FUNCTION_BLOCK PUBLIC FB_AirConditioning
VAR_OUTPUT
	bActive			: BOOL;
	lrTemperature	: LREAL;
END_VAR

METHOD PUBLIC Activate
bActive := TRUE;
END_METHOD

PROPERTY PUBLIC Activated : BOOL
GET
Activated := bActive;
END_GET
END_PROPERTY

METHOD PUBLIC Deactivate
bActive := false;
END_METHOD

METHOD PUBLIC SetTemperature : BOOL
VAR_INPUT
	lrNewTemperature	: LREAL;
END_VAR
lrTemperature := lrNewTemperature;
END_METHOD

PROPERTY PUBLIC Temperature : LREAL
GET
Temperature := lrTemperature;
END_GET
END_PROPERTY

END_FUNCTION_BLOCK

(* stored: Version 1.1.0.1, ProductVersion 3.1.4024.12
   POU FB_AirConditioning: Id {33062600-9863-4605-87a9-22af9fa61198}, SpecialFunc None
   Method Activate: Id {c8dc9767-89fe-4d6f-b741-d4ab544ed8ab}
   Property Activated: Id {21e3bc8a-4876-47a7-afea-a4e10750785d}
   Get Get: Id {680c8b23-0885-4341-95b1-03a3294e2c73}
   Method Deactivate: Id {56e8a2df-9631-413f-ba89-ee0d5381af93}
   Method SetTemperature: Id {ebb842b8-5199-490c-ace8-ece186a9f51e}
   Property Temperature: Id {91264303-577d-45f7-89af-7cf532fe6a67}
   Get Get: Id {463db962-a01c-4a3b-a8ab-7f75eeb1e2ad} *)
